(* Logix 5000 project; controller Transcat_L33ER vendor 1 type 14 code 107 rev 32.11; software revision 32.02 *)
// Upgraded CPLX to handle up to 32 EIP Nodes

TASK MainTask (continuous, watchdog 500 ms) : MainProgram

MODULES
   Local : vendor 1 type 14 code 107 (Compact 0, rev 32.11)
      GF201_Bentonite_Feeder : PowerFlex 525-EENET (Ethernet 192.168.1.195, rev 5.1, Output RPI 20 ms)   // Thayer Weigh Belt Feeder
      MX101_UpperHowesVFD : PowerFlex 525-EENET (Ethernet 192.168.1.191, rev 5.1, Output RPI 20 ms)   // VFD for Upper Howes Mixer
           MX101_UpperHowesVFD:I.Faulted   // UpperHowes Drive Faulted
           MX101_UpperHowesVFD:I.DriveStatus.4   // 1 = Accelerating
           MX101_UpperHowesVFD:I.Ready   // UpperHowes Drive Ready Status
           MX101_UpperHowesVFD:I.DriveStatus.10   // 1 - parameter locked
           MX101_UpperHowesVFD:I.DriveStatus.1   // 1 = Running, 0 - Stopped
           MX101_UpperHowesVFD:I.Active   // UpperHowes Drive Active
           MX101_UpperHowesVFD:I.DriveStatus.0   // 1 = Drive is Ready
           MX101_UpperHowesVFD:I.DriveStatus.8   // 1 = At Referecne Speed
           MX101_UpperHowesVFD:I.DriveStatus.3   // 1 = Rotating Forward
           MX101_UpperHowesVFD:I.DriveStatus.5   // 1= Decelerating
           MX101_UpperHowesVFD:I.DriveStatus.6   // not used
           MX101_UpperHowesVFD:I.DriveStatus.9   // 1 - Main Freq by Active Comms
           MX101_UpperHowesVFD:I.DriveStatus.7   // 1= Faulted
           MX101_UpperHowesVFD:I.DriveStatus.2   // 1 = Forward, 0 = Reverse
           MX101_UpperHowesVFD:O.Stop   // Drive Stop
           MX101_UpperHowesVFD:O.Start   // Drive Start
           MX101_UpperHowesVFD:O.FreqCommand   // Input Hz into Source A: 0-60 Hz range
      VF101_Medium_Feeder : PowerFlex 525-EENET (Ethernet 192.168.1.196, rev 5.1, Output RPI 20 ms)   // Medium Feeder
      MX201_LowerHowesVFD : PowerFlex 525-EENET (Ethernet 192.168.1.192, rev 5.1, Output RPI 20 ms)   // VFD for Lower Howes Mixer
           MX201_LowerHowesVFD:I.Faulted   // LowerHowes Drive Faulted
           MX201_LowerHowesVFD:I.Ready   // LowerHowes Drive Ready Status
           MX201_LowerHowesVFD:I.Active   // LowerHowes Drive Active
           MX201_LowerHowesVFD:O.Stop   // Drive Stop
      VF201_Small_Feeder_2 : PowerFlex 525-EENET (Ethernet 192.168.1.197, rev 5.1, Output RPI 20 ms)   // Acrison Small Feeder 2
      SBC2000_1_Acrison : ETHERNET-MODULE (Ethernet 192.168.1.150, rev 1.1, Output RPI 250 ms)   // Acrison Drive 1 to control Small Feeder 1
           SBC2000_1_Acrison:I.Data   // Ethernet Input Array
           SBC2000_1_Acrison:I.Data[1]   // PV - Feedrate - kg/hr
           SBC2000_1_Acrison:I.Data[2]   // Totalizer 1 - kg
           SBC2000_1_Acrison:I.Data[0]   // SP-FeedRate - kg/hr
           SBC2000_1_Acrison:I.Data[4]   // Hopper Level - %
           SBC2000_1_Acrison:I.Data[3]   // OT - Motor Speed - %
           SBC2000_1_Acrison:O.Data[15]   // When Command_Bits is 1, machine is running.
      Thayer1_BS : ETHERNET-MODULE (Ethernet 192.168.1.140, rev 1.1, Output RPI 50 ms)   // Thayer 1 Weight Belt Feeder
      Thayer2_BS : ETHERNET-MODULE (Ethernet 192.168.1.160, rev 1.1, Output RPI 50 ms)   // Thayer 2 Weigh Belt Feeder
      XS26_PLC_Safety_Controller : XS26 SC26 SC10 (Ethernet 192.168.1.211, rev 2.1, StandardDataDriven RPI 100 ms)   // XS26 Safety Controller in PLC cabinet
      XS26_VFD_Cabinet_Safety_Controller : XS26 SC26 SC10 (Ethernet 192.168.1.212, rev 2.1, StandardDataDriven RPI 100 ms)   // Banner XS26 Safety Controller with 3 expansion modules in VFD cabinet
      TC_Remote_IO : 1734-AENT (Ethernet 192.168.1.190, rev 6.1, Output RPI 20 ms)
         TC_8Pt_Analog_Input : vendor 1 type 115 code 210 (PointIO 1, rev 3.1, Input RPI 80 ms)
         TC_8pt_DC_Input_Sink : 1734-IB8 (PointIO 2, rev 3.1)
         TC_8pt_Digital_Output_Sourced : 1734-OB8 (PointIO 3, rev 3.1)
         TC_4pt_Relay_Output : 1734-OW4 (PointIO 4, rev 3.1)
END_MODULES

TYPE Acrison_Feeder :   // Acrison Feeder Tags
STRUCT
   AutoMan : BOOL;   // On - Auto Control - follows AutoRun bit, Off - Manaul Control - follows Manual Run bit
   ManualRun : BOOL;   // On - Runs feeder in Manual, Off - Stops feeder in manual
   AutoRun : BOOL;   // On - Runs feeder in Auto Off - Stops feeder in Auto
   Interlock : BOOL;   // Interlock bit - if on - Feeder will not run
   Output : BOOL;   // On - Feeder runs, Off Feeder stops
   Int_Status : DINT;   // 32 Status bits from feeder
   SP_HMI : REAL;   // setpoint from HMI
   SP_READ : REAL;   // setpoint read back from controller
   Enable : BOOL;   // Enable logic to run feeder
   OT_Actual_Hz : REAL;   // The current output of the VFD in Hz
   FreqHz_Real : REAL;   // The command frequency of the drive in Hz
   CycleTime : TIMER;   // running time of current cycle
   CampTime : TIMER;   // running time of current campaign / batch
   TotalTime : TIMER;   // total time the device / motor has run since last reset
   OneShots : BOOL[32];   // 32 Booleans to hold one-shots assicated with this device
   TimeRunTarget : DINT;   // Target Amount of time in seconds to run the device
   StartDelay : TIMER;   // Delay before motor start
   StartDelayms : DINT;   // Start delay in milliseconds
   TimeRunStart : BOOL;   // Bit to start and run a timed run
END_STRUCT
END_TYPE

TYPE BronkhorstFlowMeter :   // Read and write values for Bronkhorst Flow Meters
STRUCT
   SP_R : REAL;   // Set Point - FlowRate - Read - g/min - read from Flow Meter
   PV_R : REAL;   // Process Variable - FlowRate - Read - g/min
   OT_R : REAL;   // Output - PumpSpeed - Read - %
   TempC : REAL;   // Temperaure - Read - Deg C
   Density : REAL;   // Density - Read - g/liter
   Usertag : STRING;   // User Tag in Flow Meter - String
   FBNode : INT;   // Flow Bus Node # - Integer
   Model : STRING;   // Flow Meter Model #
   Serial : STRING;   // Flow Meter Serial #
   Capacity : REAL;   // Max Flow Rate of Flow Meter
   Enable : BOOL;   // Device enable bit
   AutoMan : BOOL;   // Select Auto / Manual Mode
   AutoRun : BOOL;   // On / Off in Auto Mode
   ManualRun : BOOL;   // On / Off- in Manual Mode
   Interlock : BOOL;   // Interlock Bit
   Output : BOOL;   // Output Bit for Device
   SP_HMI : REAL;   // Setpoint from HMI
   SP_W : REAL;   // Setpoint - flowrate g/min - write to Flow Meter from PLC
   Connected : BOOL;   // Is flow meter connecte to the flow bus network
   Alarm : BOOL;   // Alarm Bit - if on flow meter in ALarm Status
   Running : BOOL;   // the flow meter is running / dosing
   AlarmReset : BOOL;   // bit to toggle to reset alarm
   AlarmID : INT;   // Integer # that describes the type of Alarm
   ReadTime : INT;   // time in milliseconds to read the flow meter data
   DevPct : REAL;   // % deviation of process variable from setpoint
   CycleTime : TIMER;   // running time of current cycle
   CampTime : TIMER;   // running time of current campaign
   TotalTime : TIMER;   // total time the device / motor has run since last reset
   OneShots : BOOL[32];   // 32 Booleans to hold one-shots assicated with this device
   TimeRunTarget : DINT;   // Target Amount of time in seconds to run the device
   StartDelay : TIMER;   // Delay before motor start
   StartDelayms : DINT;   // Start delay in milliseconds
   TimeRunStart : BOOL;   // Bit to start and run a timed run
   Totalizer : REAL;   // Total dosed by flow meter since last reset
   TotalizerReset : BOOL;   // Bit to reset the totalizer (called a counter in Bronkhorst literature)
   TotalizerEnable : BOOL;   // Bit to turn the totalizer on / off
END_STRUCT
END_TYPE

TYPE Device :   // this UDT will be the template for all equipment / devices - feeders, flow meters, others and will be set up for each device to be indexed and processed via indirect addressing
STRUCT
   SP_R : REAL;   // Set Point - FlowRate - Read - g/min - read from Flow Meter
   PV_R : REAL;   // Process Variable - FlowRate - Read - g/min
   OT_R : REAL;   // Output - PumpSpeed - Read - %
   TempC : REAL;   // Temperaure - Read - Deg C
   Density : REAL;   // Density - Read - g/liter
   Usertag : STRING;   // User Tag in Flow Meter - String
   FBNode : INT;   // Flow Bus Node # - Integer
   Model : STRING;   // Flow Meter Model #
   Serial : STRING;   // Flow Meter Serial #
   Capacity : REAL;   // Max Flow Rate of Flow Meter
   Enable : BOOL;   // Device enable bit
   AutoMan : BOOL;   // Select Auto / Manual Mode
   AutoRun : BOOL;   // On / Off in Auto Mode
   ManualRun : BOOL;   // On / Off- in Manual Mode
   Interlock : BOOL;   // Interlock Bit
   Output : BOOL;   // Output Bit for Device
   SP_HMI : REAL;   // Setpoint from HMI
   SP_W : REAL;   // Setpoint - flowrate g/min - write to Flow Meter from PLC
   Connected : BOOL;   // Is flow meter connecte to the flow bus network
   Alarm : BOOL;   // Alarm Bit - if on flow meter in ALarm Status
   Running : BOOL;   // the flow meter is running / dosing
   AlarmReset : BOOL;   // bit to toggle to reset alarm
   AlarmID : INT;   // Integer # that describes the type of Alarm
   ReadTime : INT;   // time in milliseconds to read the flow meter data
   DevPct : REAL;   // % deviation of process variable from setpoint
   CycleTime : TIMER;   // running time of current cycle
   CampTime : TIMER;   // running time of current campaign
   TotalTime : TIMER;   // total time the device / motor has run since last reset
   OneShots : BOOL[32];   // 32 Booleans to hold one-shots assicated with this device
   TimedRunTarget : DINT;   // Target Amount of time in seconds to run the device
   StartDelay : TIMER;   // Delay before motor start
   StartDelayms : DINT;   // Start delay in milliseconds
   TimeRunEnable : BOOL;   // Bit to enable / activate a timed (campaign timed) run
   Totalizer : REAL;   // Total dosed by flow meter since last reset
   TotalizerReset : BOOL;   // Bit to reset the totalizer (called a counter in Bronkhorst literature)
   TotalizerEnable : BOOL;   // Bit to turn the totalizer on / off
   TimedRunTargetms : DINT;   // Timed run target convered to ms for use in timers
   OutPutTest : BOOL;   // A bit to simulate output that does NOT control anything
   StartDelay_ST_Timer : FBD_TIMER;   // Start delay timer to use in stuctured text
   PermissivesAuto : BOOL;   // Bit to allow device to start in AUTO as long as all permissive conditions met
   PermissivesMan : BOOL;   // Bit to allow device to start in Manual as long as all permissive conditions met
   Error : REAL;   // % Error from SP (Positive Value = running above SP and vice versa)
   ErrorTimer : TIMER;   // Amont of consecutive seconds the Error is permitterd to be out of range (+/- x%) before triggering interlock
   ErrorLimit : REAL;   // + / - % error range the system can operate in
END_STRUCT
END_TYPE

TYPE Howes_Mixer :   // Howes Mixer Tags
STRUCT
   AutoMan : BOOL;   // On - Auto Control - follows AutoRun bit, Off - Manaul Control - follows Manual Run bit
   ManualRun : BOOL;   // On - Runs feeder in Manual, Off - Stops feeder in manual
   AutoRun : BOOL;   // On - Runs feeder in Auto Off - Stops feeder in Auto
   Interlock : BOOL;   // Interlock bit - if on - Feeder will not run
   Output : BOOL;   // On - Feeder runs, Off Feeder stops
   Int_Status : DINT;   // 32 Status bits from feeder
   SP_HMI : REAL;   // setpoint from HMI
   SP_READ : REAL;   // setpoint read back from controller
   Enable : BOOL;   // Enable logic to run mixer
   FreqHz_Real : REAL;   // Frequency in Hz expressed as real #
   OT_Actual_Hz : REAL;   // The current output of the drive in Hz
   CycleTime : TIMER;   // currnet cycle run time
   CampTime : TIMER;   // current campaign run time
   TotalTime : TIMER;   // total run time since last reset
   OneShots : BOOL[32];   // 32 Booleans to hold one shots associated with this device
   TimeRunTarget : DINT;   // Target Amount of time in seconds to run the device
   TimeRunStart : BOOL;   // Bit to start and run a timed run
   StartDelay : TIMER;   // Delay before motor starts
   StartDelayms : DINT;   // Delay before motor starts in milliseconds
   RPM : REAL;   // RPM from speed sensor
END_STRUCT
END_TYPE

TYPE Thayer_WB_Feeder :   // Thayer WB Feeder Tags
STRUCT
   AutoMan : BOOL;   // On - Auto Control - follows AutoRun bit, Off - Manaul Control - follows Manual Run bit
   ManualRun : BOOL;   // On - Runs feeder in Manual, Off - Stops feeder in manual
   AutoRun : BOOL;   // On - Runs feeder in Auto Off - Stops feeder in Auto
   Interlock : BOOL;   // Interlock bit - if on - Feeder will not run
   Output : BOOL;   // On - Feeder runs, Off Feeder stops
   Int_Status : DINT;   // 32 Status bits from feeder
   SP_HMI : REAL;   // setpoint from HMI
   SP_READ : REAL;   // setpoint read back from controller
   Enable : BOOL;   // Enable logic to run feeder
   CycleTime : TIMER;   // current cycle run time
   CampTime : TIMER;   // current campaing run time
   TotalTime : TIMER;   // total run time since last reset
   OneShots : BOOL[32];   // 32 Booleans to hold one-shots assicated with this device
   TimeRunTarget : DINT;   // Target Amount of time in seconds to run the device - from recipe
   StartDelay : TIMER;   // Delay before starting motor / equipment
   StartDelayms : DINT;   // Start delay in milliseconds
   TimeRunStart : BOOL;   // Bit to start and run a timed run
END_STRUCT
END_TYPE

VAR_GLOBAL   (* controller tags *)
   AcrisonFeedRateSetPoint : MESSAGE;   // Message Command to Write to Feed Rate Set Point in Acrison from GF103.SP_HMI in kg/hr
        MessageParameters(ServiceCode := 16#0010, LocalElement := GF301.SP_HMI, ...)
   AllDevice1stScanDone : BOOL := 1;   // When this bit is set - all devices have been scanned once and bits reset
   AllDeviceEnable : BOOL := 1;   // A bit to enable or disable the running of all devices
   AllReset : BOOL;   // Bit to reset Auto/Man, AutoRun, RecipeRun, TimedRunEnable to 0 from PLC
   alwaysOFF : BOOL;
   AlwaysOFF2 : BOOL;
   AlwaysOn : BOOL;
   AnyAutoRun : BOOL;   // Bit that in on if ANY device is placed into Auto run (to signal pre-start beed)
   AnyAutoRunFlag : BOOL;   // A flag that indicates if any device is in Auto Run (used with pre-start beep logic)
   AnyManRunFlag : BOOL;   // A flag that indicates if any device is in Manual Run (used with pre-start beep logic)
   AnyManualRun : BOOL;   // Bit that in on if ANY device is placed into manual run (to signal pre-start beed)
   AnyRun : BOOL := 1;   // Bit that is true if any Maunal Run or Auto Run bit is set
   AnyRunFlag : BOOL;   // A Flag to know if any device in already running in Auto or Manual
   BeaconBeepAlarm : BOOL;   // Beep Alarm
   BeaconBlueLight : ALIAS FOR TC_Remote_IO:3:O.3;   // Blue Beacon Light
   BeaconGreenLight : ALIAS FOR TC_Remote_IO:3:O.2;   // Green Beacon Light
   BeaconRedLight : ALIAS FOR TC_Remote_IO:3:O.0;   // Red Beacon Light
   BeaconYellowLight : ALIAS FOR TC_Remote_IO:3:O.1;   // Yellow Beacon Light
   Beep : BOOL;   // Bit to Activte Beacon Alarm
   BeepNew : ALIAS FOR TC_Remote_IO:3:O.4;
   Device : Device[20] := ([0].SP_HMI := 10.6, [0].CycleTime.PRE := 288000000, [0].CycleTime.ACC := 731171, [0].CampTime.PRE := 288000000, [0].CampTime.ACC := 20003, [0].TotalTime.PRE := 288000000, [0].TotalTime.ACC := 11616964, [0].OneShots[4] := 1, [0].TimedRunTarget := 20, [0].StartDelay.PRE := 2000, [0].StartDelayms := 2, [0].TimedRunTargetms := 20000, [0].StartDelay_ST_Timer.TimerEnable := 1, [0].StartDelay_ST_Timer.PRE := 10000, [0].ErrorTimer.PRE := 10000, [1].SP_HMI := 10.6, [1].CycleTime.PRE := 288000000, [1].CycleTime.ACC := 730212, [1].CampTime.PRE := 288000000, [1].CampTime.ACC := 20004, [1].TotalTime.PRE := 288000000, [1].TotalTime.ACC := 7079420, [1].OneShots[4] := 1, [1].TimedRunTarget := 20, [1].StartDelay.PRE := 2000, [1].StartDelayms := 2, [1].TimedRunTargetms := 20000, [1].ErrorTimer.PRE := 60000, [2].CycleTime.PRE := 288000000, [2].CycleTime.ACC := 173670, [2].CampTime.PRE := 288000000, [2].CampTime.ACC := 5003, [2].TotalTime.PRE := 288000000, [2].TotalTime.ACC := 2719384, [2].OneShots[4] := 1, [2].TimedRunTarget := 5, [2].StartDelay.PRE := 2000, [2].StartDelayms := 2, [2].TimedRunTargetms := 5000, [2].PermissivesAuto := 1, [2].PermissivesMan := 1, [3].CycleTime.PRE := 288000000, [3].CycleTime.ACC := 2659, [3].CampTime.PRE := 288000000, [3].TotalTime.PRE := 288000000, [3].TotalTime.ACC := 109408498, [3].OneShots[4] := 1, [3].TimedRunTarget := 10, [3].StartDelay.PRE := 2000, [3].StartDelayms := 2, [3].TimedRunTargetms := 10000, [3].PermissivesAuto := 1, [3].PermissivesMan := 1, [4].CycleTime.PRE := 288000000, [4].CycleTime.ACC := 79705, [4].CampTime.PRE := 288000000, [4].TotalTime.PRE := 288000000, [4].TotalTime.ACC := 440481, [4].OneShots[4] := 1, [4].StartDelay.PRE := 2000,
        [4].StartDelayms := 2, [4].PermissivesAuto := 1, [4].PermissivesMan := 1, [5].CycleTime.PRE := 288000000, [5].CycleTime.ACC := 174455, [5].CampTime.PRE := 288000000, [5].CampTime.ACC := 39951, [5].TotalTime.PRE := 288000000, [5].TotalTime.ACC := 3397807, [5].OneShots[4] := 1, [5].TimedRunTarget := 120, [5].StartDelay.PRE := 2000, [5].StartDelayms := 2, [5].TimedRunTargetms := 120000, [5].PermissivesAuto := 1, [5].PermissivesMan := 1, [6].CycleTime.PRE := 288000000, [6].CycleTime.ACC := 485, [6].CampTime.PRE := 288000000, [6].CampTime.ACC := 39952, [6].TotalTime.PRE := 288000000, [6].TotalTime.ACC := 3344121, [6].OneShots[4] := 1, [6].TimedRunTarget := 120, [6].StartDelay.PRE := 2000, [6].StartDelayms := 2, [6].TimedRunTargetms := 120000, [6].PermissivesAuto := 1, [6].PermissivesMan := 1, [7].SP_HMI := 150.0, [7].CycleTime.PRE := 288000000, [7].CycleTime.ACC := 39946, [7].CampTime.PRE := 288000000, [7].CampTime.ACC := 39951, [7].TotalTime.PRE := 288000000, [7].TotalTime.ACC := 8389325, [7].OneShots[4] := 1, [7].TimedRunTarget := 120, [7].StartDelay.PRE := 5000, [7].StartDelayms := 5, [7].TimedRunTargetms := 120000, [8].CycleTime.PRE := 288000000, [8].CycleTime.ACC := 39947, [8].CampTime.PRE := 288000000, [8].CampTime.ACC := 39952, [8].TotalTime.PRE := 288000000, [8].TotalTime.ACC := 7574006, [8].OneShots[4] := 1, [8].TimedRunTarget := 120, [8].StartDelay.PRE := 5000, [8].StartDelayms := 5, [8].TimedRunTargetms := 120000, [9].CycleTime.PRE := 288000000, [9].CycleTime.ACC := 39946, [9].CampTime.PRE := 288000000, [9].CampTime.ACC := 39951, [9].TotalTime.PRE := 288000000, [9].TotalTime.ACC := 6215395, [9].OneShots[4] := 1, [9].TimedRunTarget := 120,
        [9].StartDelay.PRE := 5000, [9].StartDelayms := 5, [9].TimedRunTargetms := 120000, [10].CycleTime.PRE := 288000000, [10].CampTime.PRE := 288000000, [10].TotalTime.PRE := 288000000, [10].OneShots[2] := 1, [10].OneShots[4] := 1, [11].CycleTime.ACC := 6, [11].CycleTime.DN := 1, [11].TotalTime.ACC := 7, [11].TotalTime.DN := 1, [11].OneShots[4] := 1, [11].PermissivesAuto := 1, [11].PermissivesMan := 1);
        [8]   // FT104 - Bronkhorst Water Dosing System
        [9]   // FT105 Bronkhorst Fragrance Dosing System
        [4]   // GF301 Small Feeder - Acrison LIW
        [0]   // MX101 - Upper Howes Mixer
        [1]   // MX201 - Lower Howes Mixer
        [2]   // GF101 - Thayer1 WB Feeder
        [3]   // GF201 - Thayer2 WB Feeder
        [5]   // VF101 Medium Feeder - Acurate
        [7]   // FT103 - Bronkhorst Oil Dosing System
        [6]   // VF201 Small Feeder 2 - Acrison
   DINT_Temp : DINT;   // Place to hold Dint's durng transition to new PLC
   DiscreteTemp : BOOL;   // A temporay boolean to hold positions during PLC transer
   dNum : INT := 1;   // The index of the current device being processed
   DoseCounter : COUNTER := (ACC := 522, CU := 1, DN := 1);   // Counts the # of doses since last reset
   DoseCounterReset_HMI : BOOL;   // HMI bit to reset the dose counter
   DoseStart : BOOL;   // Bit to start dosing sequence
   DoseStartOneShot : BOOL := 1;   // One shot to start dosing
   DoseStop : BOOL;   // Bit to stop dosing
   DoseStopOneShot : BOOL := 1;   // one shot to stop dosing
   DoseTarget : REAL := 27.9;   // Target dose amount
   FT103 : BronkhorstFlowMeter := (Usertag := 'FT-103', Model := 'M55-RGD-25-0-S', Serial := 'M22213015A', Capacity := 1000.00006, Enable := 1, SP_HMI := 50.0, ReadTime := 500, CycleTime.PRE := 288000000, CycleTime.ACC := 19487, CampTime.PRE := 28800000, CampTime.ACC := 10001, TotalTime.PRE := 999999999, TotalTime.ACC := 114629);
   FT104 : BronkhorstFlowMeter := (PV_R := -97.77293, TempC := 21.284956, Density := 9999.0, Usertag := 'FT-104          ', Model := 'M55-RGD-25-0-S', Serial := 'M22213015C', Capacity := 10000.0, Enable := 1, SP_HMI := 100.0, Connected := 1, ReadTime := 70, CycleTime.PRE := 288000000, CycleTime.ACC := 3248, CampTime.PRE := 28800000, CampTime.ACC := 10001, TotalTime.PRE := 999999999, TotalTime.ACC := 84417, StartDelay.PRE := 2000, StartDelayms := 2);
   FT105 : BronkhorstFlowMeter := (PV_R := 0.458107, TempC := 28.406788, Density := 4.5310874, Usertag := 'FT-105          ', Model := 'M14-RGD-22-0-S', Serial := 'M20210127A', Capacity := 202.79999, Enable := 1, SP_HMI := 75.0, Connected := 1, ReadTime := 64, CycleTime.PRE := 288000000, CycleTime.ACC := 11357, CampTime.PRE := 28800000, CampTime.ACC := 10001, TotalTime.PRE := 999999999, TotalTime.ACC := 55929, StartDelay.PRE := 4000, StartDelayms := 4);
   GF101 : Thayer_WB_Feeder := (SP_HMI := 21.4, SP_READ := 21.375, Enable := 1, CycleTime.PRE := 288000000, CycleTime.ACC := 9195, CampTime.PRE := 28800000, CampTime.ACC := 10001, TotalTime.PRE := 999999999, TotalTime.ACC := 1761327, StartDelay.PRE := 2000, StartDelayms := 2);   // Thayer 1 Tags
   GF101_Alarm_ExcessDevSP : ALIAS FOR Thayer1_BS:I.Data[8].7;   // Thayer 1 (GF101) - Alarm - excessive deviation from SP
   GF101_LoadCell : ALIAS FOR Thayer1Data[15];   // Thayer 1 (GF101) load cell in lbs
   GF101_LoadCellTempF : ALIAS FOR Thayer1Data[16];   // Thayer 1 (GF101) load cell temperature in Deg F
   GF101_OutputPct : ALIAS FOR Thayer1Data[5];   // Thayer 1 (GF101) Output to motor in pct - raw
   GF101_RunningLoad : ALIAS FOR Thayer1Data[0];   // Thayer 1 (GF101) Running Load - current load on belt in lbs
   GF101_RunningRate : ALIAS FOR Thayer1Data[1];   // Thayer 1 (GF101) Running Rate - current PV displayed on the operator screen
   GF101_RunningSpeed : ALIAS FOR Thayer1Data[2];   // Thayer 1 (GF101) Running Soeed - current speed of the belt in ft/min?
   GF101_SetPoint : ALIAS FOR Thayer1Data[3];   // Thayer 1 (GF101) SetPoint - in lb/min
   GF101_Shutdown_ExcessDevSp : ALIAS FOR Thayer1_BS:I.Data[10].7;   // Thayer 1 (GF101) - Shutdown - excessive deviation from SP
   GF101_Status_AutoMan : ALIAS FOR Thayer1_BS:I.Data[0].1;   // Thayer 1 (GF101) - Auto / Manual Status - 1 = Auto 0 = Manual
   GF101_Status_Coasting : ALIAS FOR Thayer1_BS:I.Data[0].2;   // Thayer 1 (GF101) - Coasting to stop of shutdown - 1 = Coasting, 0 = Not coasting
   GF101_Status_EchoBack : ALIAS FOR Thayer1_BS:I.Data[0].13;   // Thayer 1 (GF101) - Echo back bit
   GF101_Status_HeartBeat : ALIAS FOR Thayer1_BS:I.Data[0].14;   // Thayer 1 (GF101) - HeartBeat - every 5 seconds
   GF101_Status_Interlocked : ALIAS FOR Thayer1_BS:I.Data[0].8;   // Thayer 1 (GF101) - Interlocked Bit - 1 = Interlocked 0 = Not Interlocked
   GF101_Status_RunStop : ALIAS FOR Thayer1_BS:I.Data[0].0;   // Thayer 1 (GF101) - Operating Status - 1 = Running 0 = Stopped
   GF101_Status_TachGT0 : ALIAS FOR Thayer1_BS:I.Data[0].9;   // Thayer 1 (GF101) - 1 = Tachometer > 0 0 = Tachometer = 0
   GF101_TachHz : ALIAS FOR Thayer1Data[14];   // Thayer 1 (GF101) Tachometer in Hz
   GF101_Totalizer1 : ALIAS FOR Thayer1Data[9];   // Thayer 1 (GF101) Totalizer 1 in lbs
   GF101_Totalizer2 : ALIAS FOR Thayer1Data[10];   // Thayer 1 (GF101) Totalizer 2 in lbs
   GF101_Write_Acknowledge : ALIAS FOR Thayer1_BS:O.Data[2].5;   // Thayer 1 (GF101) Acknowledge
   GF101_Write_AutoMan : ALIAS FOR Thayer1_BS:O.Data[0].1;   // Thayer 1 (GF101) Auto / Manual 1 = Auto 2 = Manual
   GF101_Write_RunStop : ALIAS FOR Thayer1_BS:O.Data[0].0;   // Thayer 1 (GF101) 1 = Run / 0 = off/stop
   GF101_Write_Total1Reset : ALIAS FOR Thayer1_BS:O.Data[2].1;   // Thayer 1 (GF101) Totalizer 1 reset
   GF101_Write_Total2Reset : ALIAS FOR Thayer1_BS:O.Data[2].2;   // Thayer 1 (GF101) Totalizer 2 reset
   GF101OutpuyPct1sec : ALIAS FOR Thayer1Data[6];   // Thayer 1 (GF101) Output to motor in pct - averaged over 1 sec
   GF201 : Thayer_WB_Feeder := (SP_HMI := 20.0, SP_READ := 20.0, Enable := 1, CycleTime.PRE := 288000000, CycleTime.ACC := 17126, CampTime.PRE := 28800000, CampTime.ACC := 10001, TotalTime.PRE := 999999999, TotalTime.ACC := 1645614, StartDelay.PRE := 2000, StartDelayms := 2);   // Thayer 2 Tags
   GF201_Alarm_ExcessiDevSP : ALIAS FOR Thayer2_BS:I.Data[8].7;   // Thayer 2 (GF201) - Alarm - excessive deviation from SP
   GF201_LoadCell : ALIAS FOR Thayer2Data[15];   // Thayer 2 (GF201) load cell in lbs
   GF201_LoadCellTempF : ALIAS FOR Thayer2Data[16];   // Thayer 2 (GF201) load cell temperature in Deg F
   GF201_OutputPct : ALIAS FOR Thayer2Data[5];   // Thayer 2 (GF201) Output to motor in pct - raw
   GF201_RunningLoad : ALIAS FOR Thayer2Data[0];   // Thayer 2 (GF201) Running Load - current load on belt in lbs
   GF201_RunningRate : ALIAS FOR Thayer2Data[1];   // Thayer 2 (GF201) Running Rate - current PV displayed on the operator screen
   GF201_RunningSpeed : ALIAS FOR Thayer2Data[2];   // Thayer 2 (GF201) Running Soeed - current speed of the belt in ft/min?
   GF201_SetPoint : ALIAS FOR Thayer2Data[3];   // Thayer 2 (GF201) SetPoint - in lb/min
   GF201_Shutdown_ExcessDevSP : ALIAS FOR Thayer2_BS:I.Data[10].7;   // Thayer 2 (GF201) - Shutdown - excessive deviation from SP
   GF201_Status_AutoMan : ALIAS FOR Thayer2_BS:I.Data[0].1;   // Thayer 2 (GF201) - Auto / Manual Status - 1 = Auto 0 = Manual
   GF201_Status_Coasting : ALIAS FOR Thayer2_BS:I.Data[0].2;   // Thayer 2 (GF201) - Coasting to stop of shutdown - 1 = Coasting, 0 = Not coasting
   GF201_Status_EchoBack : ALIAS FOR Thayer2_BS:I.Data[0].13;   // Thayer 2 (GF201) - Echo back bit
   GF201_Status_HeartBeat1 : ALIAS FOR Thayer2_BS:I.Data[0].14;   // Thayer 2 (GF201) - HeartBeat - every 5 seconds
   GF201_Status_Interlocked : ALIAS FOR Thayer2_BS:I.Data[0].8;   // Thayer 2 (GF201) - Interlocked Bit - 1 = Interlocked 0 = Not Interlocked
   GF201_Status_RunStop : ALIAS FOR Thayer2_BS:I.Data[0].0;   // Thayer 2 (GF201) - Operating Status - 1 = Running 0 = Stopped
   GF201_Status_TachGT0 : ALIAS FOR Thayer2_BS:I.Data[0].9;   // Thayer 2 (GF201) - 1 = Tachometer > 0 0 = Tachometer = 0
   GF201_TachHz : ALIAS FOR Thayer2Data[14];   // Thayer 2 (GF201) Tachometer in Hz
   GF201_Totalizer1 : ALIAS FOR Thayer2Data[9];   // Thayer 2 (GF201) Totalizer 1 in lbs
   GF201_Totalizer2 : ALIAS FOR Thayer2Data[10];   // Thayer 2 (GF201) Totalizer 2 in lbs
   GF201_Write_Acknowledge : ALIAS FOR Thayer2_BS:O.Data[2].5;   // Thayer 2 (GF201) Acknowledge
   GF201_Write_AutoMan : ALIAS FOR Thayer2_BS:O.Data[0].1;   // Thayer 2 (GF201) Auto / Manual 1 = Auto 2 = Manual
   GF201_Write_RunStop : ALIAS FOR Thayer2_BS:O.Data[0].0;   // Thayer 2 (GF201) 1 = Run / 0 = off/stop
   GF201_Write_Total1Reset : ALIAS FOR Thayer2_BS:O.Data[2].1;   // Thayer 2 (GF1201) Totalizer 1 reset
   GF201_Write_Total2Reset : ALIAS FOR Thayer2_BS:O.Data[2].2;   // Thayer 2 (GF201) Totalizer 2 reset
   GF201OutpuyPct1sec : ALIAS FOR Thayer2Data[6];   // Thayer 2 (GF201) Output to motor in pct - averaged over 1 sec
   GF301 : Acrison_Feeder := (Int_Status := 596060, SP_HMI := 8.0, Enable := 1, CycleTime.PRE := 288000000, CycleTime.ACC := 223848, CampTime.PRE := 28800000, CampTime.ACC := 10001, TotalTime.PRE := 999999999, TotalTime.ACC := 2086091, StartDelay.PRE := 2000, StartDelayms := 2);   // GF103 - Small Feeder 1
        .Int_Status.3   // SP Int-1 / Ext-0
        .Int_Status.5   // Batch-1 / Cont-0
        .Int_Status.11   // Alarm
        .Output   // GF103 - Acrison Small Feeder Run Bit
        .Int_Status.13   // Empty
        .Int_Status.4   // Mode - Grav-1 / Vol-0
        .Int_Status.17   // Deviation
        .Int_Status.12   // Message
        .Int_Status.14   // Overfill
        .Int_Status.15   // Acrilock
        .Int_Status.16   // No Scale
        .Int_Status.10   // Overfill / Empty
        .Int_Status.1   // Refil
        .Int_Status.2   // AutoRefill
        .Int_Status.7   // Bribble
        .Int_Status.0   // Run-1 / Stop-0
        .Int_Status.9   // Low Level
        .Int_Status.6   // Batch Complete
        .Int_Status   // 32 Bit Status Int
        .Int_Status.8   // High Level
   GF301_AlarmAck : BOOL;   // GF301 Alarm Ack Bit
   GF301_ClearCommands : BOOL;   // Bit to send clear command to GF301 command integer
   GF301_Command_Bits : INT;   // Command Word - Holds a value that gets written to Acrison SCB2000:I.Data[15] see Acrison Manual for which bits do what
        .1   // Refill Mode Man - 1 / Auto - 0
        .0   // Run-1 / Stop-0
        .8   // Setpoint - Ext -1 / Int - 0
        .2   // Batch-1 / Cont-0
        .4   // Refill ON
        .6   // Alarm Ack
        .5   // Refill OFF
        .3   // Batch Abort
        .7   // Mode Vol - 1/ Grav - 0
   GF301_IntStatus : DINT := 596060;   // 32 Bit Status INT for GF301
        .14   // Overfill
        .12   // Message
        .10   // Overfill / Empty
        .0   // Run- 1/ Stop - 0
        .15   // Acrilok
        .6   // Batch Complete
        .9   // Low Level
        .16   // No Scale
        .3   // Setpoint Int - 1 / Ext - 0
        .17   // Deviation
        .1   // Refil
        .2   // Auto Refill
        .4   // Mode Grav - 1 / Vol - 0
        .11   // Alarm
        .8   // High Level
        .13   // Empty
        .7   // Dribble
        .5   // Batch - 1 / Cont - 0
   GF301_OT : ALIAS FOR SBC2000_1_Acrison:I.Data[3];   // GF301 Ouput ot motor in %
   GF301_PV : ALIAS FOR SBC2000_1_Acrison:I.Data[1];   // GF301 PV - Process Variable
   GF301_SP_READ : ALIAS FOR SBC2000_1_Acrison:I.Data[0];   // GF301 Set point read back from Acrison - kg/min
   GF301_TOTAL : ALIAS FOR SBC2000_1_Acrison:I.Data[2];   // GF301 Totalizer in KG
   GreenFlashingOff : TIMER := (PRE := 500);
   GreenFlashingOn : TIMER := (PRE := 500);
   HertzSetting : ALIAS FOR MX101_UpperHowesVFD:O.FreqCommand.0;   // UserHzSetting
   HMI_AllReset : BOOL;   // Bit to reset Auto/Man, AutoRun, RecipeRun, TimedRunEnable to 0 from HMI
   HMI_RecipeStart : BOOL;   // Bit to start and stop recipe from HMI
   InitCount : INT := 10;   // Counter to cycle through each device on start-up and reset AutoMan, AutoRun, ManualRun bits
   MSG_FROM_SLC500 : INT[10] := ([1] := 2500, [2] := 200, [3] := 300, [4] := 400, [5] := 500, [6] := 16, [7] := 17, [8] := 18, [9] := 19); {produced}
   MX101 : Howes_Mixer := (AutoMan := 1, SP_HMI := 120.0, Enable := 1, FreqHz_Real := 40.0, CycleTime.PRE := 288000000, CycleTime.ACC := 4243, CampTime.PRE := 28800000, CampTime.ACC := 10001, TotalTime.PRE := 999999999, TotalTime.ACC := 1803981, TimeRunTarget := 10000, StartDelay.PRE := 2000, StartDelayms := 2, RPM := -0.09);
   MX101_RPM_RAW : ALIAS FOR Test_Hold;   // Raw (unscaled) RMS reading from MX101 speed sensor - RPM * 100 (range 0 - 200 RPM)
   MX101_Speed_Hold : DINT := 100;   // Constant Value for MX101 RPM meter - till Actual signal comes back from 4-20mA from sensor
   MX201 : Howes_Mixer := (AutoMan := 1, SP_HMI := 120.0, Enable := 1, FreqHz_Real := 40.0, CycleTime.PRE := 28800000, CycleTime.ACC := 117513, CampTime.PRE := 28800000, CampTime.ACC := 10001, TotalTime.PRE := 999999999, TotalTime.ACC := 1030054, TimeRunTarget := 10000, StartDelay.PRE := 2000, StartDelayms := 2, RPM := -0.06);
   MX201_RPM_RAW : ALIAS FOR Test_Hold;   // Raw (unscaled) RMS reading from MX201 speed sensor - RPM * 100 (range 0 - 200 RPM)
   MX201_Speed_Hold : DINT := 100;   // Constant Value for MX201 RPM meter - till Actual signal comes back from 4-20mA from sensor
   PowerOffThayer1 : BOOL;
   PowerOnThayer1 : BOOL;
   PT103_HP_Interlock : BOOL;
   PT103_PV_RAW : ALIAS FOR TC_Remote_IO:1:I.Ch0Data;   // Raw (unscaled) pressure reading from PT103 - PSI * 100 (range 0 - 108 PSI)
   PT104_PV_RAW : ALIAS FOR TC_Remote_IO:1:I.Ch1Data;   // Raw (unscaled) pressure reading from PT104 - PSI * 100 (range 0 - 108 PSI)
   PT105_PV_RAW : ALIAS FOR TC_Remote_IO:1:I.Ch2Data;   // Raw (unscaled) pressure reading from PT105 - PSI * 100 (range 0 - 108 PSI)
   RandomFloat : REAL[20] := ([0] := 324.0, [1] := 11268015.0, [2] := 20.713356, [3] := 16.079597, [4] := 74.3938, [5] := 86.28061, [6] := 69.73996, [7] := 47.361, [8] := 43.876316, [9] := 89.62069, [10] := 12.1234);
   RandomSeed : DINT := 258;
   RandomTimer : TIMER := (PRE := 1000, ACC := 146, EN := 1, TT := 1);
   RecipeStart : BOOL;   // Bit to start and stop a recipe execution from PLC logic
   rms : BOOL;
   StartBeepTimer : TIMER := (PRE := 2500);   // Timer to sound the beep alarm before starting a device
   TempReal1 : REAL;
   Test_Hold : DINT;   // Place for RPM and Pressure sensors to Alias for while the AI's are not available
   TestBit1 : BOOL;   // Just a test bit - does not do anything
   Thayer1_SP : REAL := 20.0;
   Thayer1Ackn_SilenceRequest : BOOL;
   Thayer1Automatic : BOOL;
   Thayer1Data : REAL[40] := ([0] := 11.25, [1] := 1.4906e-41, [3] := 21.375, [4] := 2.0, [9] := 580.0, [10] := 583.5728, [11] := 8.2028e-41, [15] := 11.25, [16] := 70.58101, [17] := 1.6071e-41, [19] := 11.25);
        [10]   // Totalizer 2
        [11]   // take a way totalizer - not used
        [2]   // Running Speed - belt speed in ft / min
        [1]   // Running Rate - Process variable in lb/min
        [7]   // not used
        [9]   // Totalizer 1
        [0]   // Running Load - load cell reading in lbs
        [15]   // Load Cell reading lbs.
        [14]   // Tachometer - Hz
        [3]   // SetPoint - in lb/min
        [8]   // not used
        [6]   // Drive Output in % (1 sec time averaged)
        [4]   // Ratio Setpoint - not used
        [5]   // Drive Output in %
        [12]   // take away belt load - not used
        [16]   // Load Cell Temperatue - Deg F
        [17]   // Auto Zero error log in %
        [13]   // Take away belt rate - not used
   Thayer1PowerOn : BOOL;
   Thayer1ResetTotalizers : BOOL;
   Thayer1SetPoint : REAL[1];
   Thayer1SpeedControl : REAL := 20.0;
   Thayer2_SP : REAL := 20.0;
   Thayer2Automatic : BOOL;
   Thayer2Data : REAL[40] := ([0] := 7.3125, [1] := 3.7907e-41, [3] := 20.0, [9] := 0.91015625, [10] := 15288.634, [11] := 7.6957e-41, [15] := 7.3125, [16] := 70.7114, [17] := 1.6071e-41, [19] := 7.3125);
   Thayer2PowerOn : BOOL;
   Thayer2ResetTotal1_HMI : BOOL;   // Bit to reset Thayer2 - totalizer 1 from HMI
   Thayer2ResetTotalizers : BOOL;
   Thayer2SpeedControl : REAL := 20.0;
   TotalRestOneShot : BOOL;   // one shot for total reset
   UHStartOneShot : BOOL;
   UHStopOneShot : BOOL;
   UpHowesHMIRun : BOOL;
   UpHowesHMIStop : BOOL;
   UpHowesSpeedHMI : INT;
   UpperHowesSpeed : INT := 2500;
   UpperHowesStart : BOOL;
   UpperHowesStop : BOOL;
   UserBit1 : BOOL;   // user controlled bit for testing
   VF101 : Acrison_Feeder := (SP_HMI := 16.81, Enable := 1, FreqHz_Real := 10.09, CycleTime.PRE := 288000000, CycleTime.ACC := 7359, CampTime.PRE := 28800000, CampTime.ACC := 10001, TotalTime.PRE := 999999999, TotalTime.ACC := 1720239, StartDelay.PRE := 5000, StartDelayms := 5);   // Medium Feeder Tags
   VF201 : Acrison_Feeder := (SP_HMI := 14.7, Enable := 1, FreqHz_Real := 8.82, CycleTime.PRE := 288000000, CycleTime.ACC := 13534, CampTime.PRE := 28800000, CampTime.ACC := 10001, TotalTime.PRE := 999999999, TotalTime.ACC := 1964985, StartDelay.PRE := 5000, StartDelayms := 5);   // Small Feeder 2 Tags
   YellowFlashOff : TIMER := (PRE := 500);
   YellowFlashOn : TIMER := (PRE := 500, ACC := 394, EN := 1, TT := 1);
   ZS101_RPM_Speed_UpperHowes : ALIAS FOR TC_Remote_IO:1:I.Ch3Data;   // Upper Howes Zero Speed Sensor RPM
   ZS102_RPM_Speed_LowerHowes : ALIAS FOR TC_Remote_IO:1:I.Ch4Data;   // Lower Howes Zero Speed Sensor RPM
END_VAR

PROGRAM MainProgram   (* main routine MainRoutine *)
VAR
   AcrisonSpeedControl : REAL := 1.0;
   AcrisonSpeedControl2 : REAL := 15.0;
   HertzInput : INT := 20;
   Int_Status : DINT := 540252;
   LowerHowesSpeedSensor : REAL := -74.971405;
   PowerOffACrison : BOOL := 1;
   PowerOnAcrison : BOOL;
   SCL_01 : SCALE := (In := -21.0, InRawMax := 16384.0, InRawMin := 3271.0, InEUMax := 300.0, Out := -75.314575, MinAlarm := 1);
   SCL_02 : SCALE := (In := -6.0, InRawMax := 16384.0, InRawMin := 3271.0, InEUMax := 300.0, Out := -74.971405, MinAlarm := 1);
   SpeedSensorUpperHowesSpeed : REAL := -75.314575;
   T1 : TIMER := (PRE := 10000);
   T2 : TIMER := (PRE := 10000, ACC := 10000, EN := 1, DN := 1);
END_VAR

ROUTINE Auxillary_Pump_AE   (* ladder *)
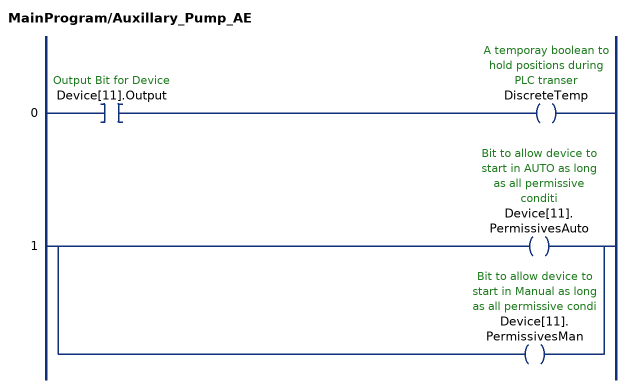
   0: XIC(Device[11].Output)OTE(DiscreteTemp);
   1: [OTE(Device[11].PermissivesAuto) ,OTE(Device[11].PermissivesMan) ];
END_ROUTINE

ROUTINE DeviceLogic   (* ladder *)
// Process the logic for each device with index and indirect addressing.
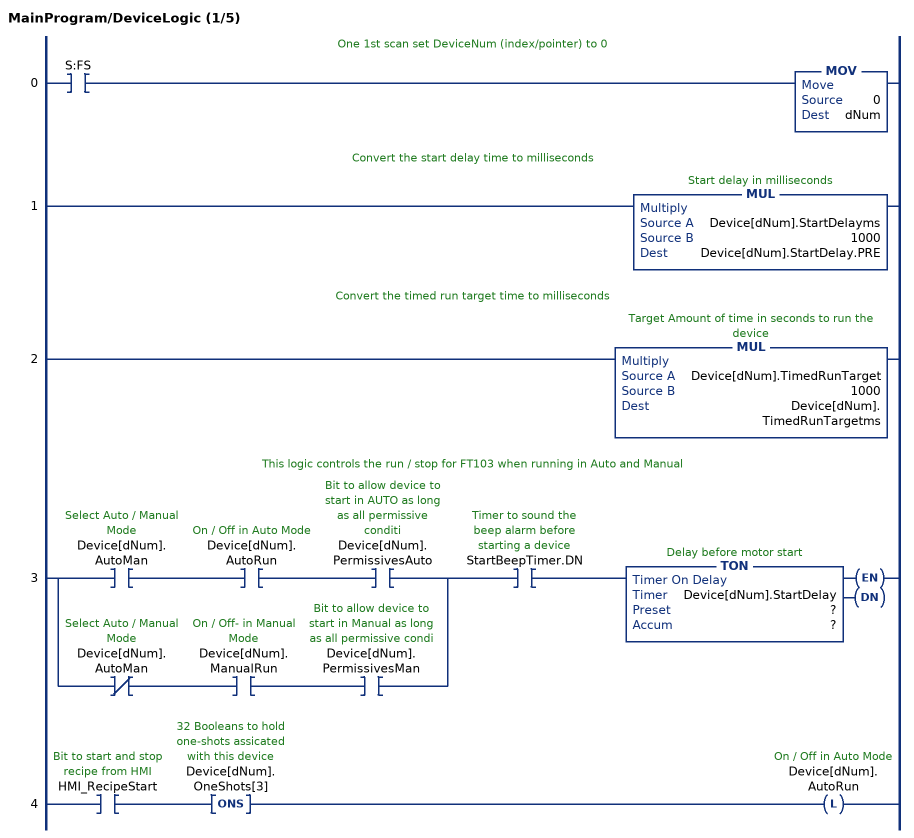
   // One 1st scan set DeviceNum (index/pointer) to 0
   0: XIC(S:FS)MOV(0,dNum);
   // Convert the start delay time to milliseconds
   1: MUL(Device[dNum].StartDelayms,1000,Device[dNum].StartDelay.PRE);
   // Convert the timed run target time to milliseconds
   2: MUL(Device[dNum].TimedRunTarget,1000,Device[dNum].TimedRunTargetms);
   // This logic controls the run / stop for FT103 when running in Auto and Manual
   3: [XIC(Device[dNum].AutoMan) XIC(Device[dNum].AutoRun) XIC(Device[dNum].PermissivesAuto) ,XIO(Device[dNum].AutoMan) XIC(Device[dNum].ManualRun) XIC(Device[dNum].PermissivesMan) ]XIC(StartBeepTimer.DN)TON(Device[dNum].StartDelay,?,?);
   4: XIC(HMI_RecipeStart)ONS(Device[dNum].OneShots[3])OTL(Device[dNum].AutoRun);
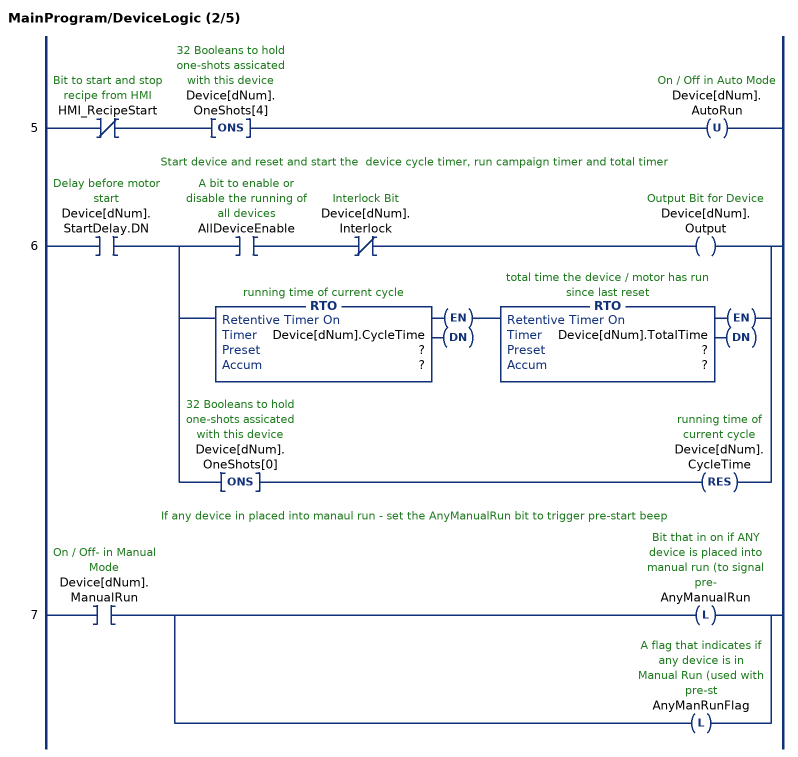
   5: XIO(HMI_RecipeStart)ONS(Device[dNum].OneShots[4])OTU(Device[dNum].AutoRun);
   // Start device and reset and start the  device cycle timer, run campaign timer and total timer
   6: XIC(Device[dNum].StartDelay.DN)[XIC(AllDeviceEnable) XIO(Device[dNum].Interlock) OTE(Device[dNum].Output) ,[RTO(Device[dNum].CycleTime,?,?) RTO(Device[dNum].TotalTime,?,?) ,ONS(Device[dNum].OneShots[0]) RES(Device[dNum].CycleTime) ] ];
   // If any device in placed into manaul run - set the AnyManualRun bit to trigger pre-start beep
   7: XIC(Device[dNum].ManualRun)[OTL(AnyManualRun) ,OTL(AnyManRunFlag) ];
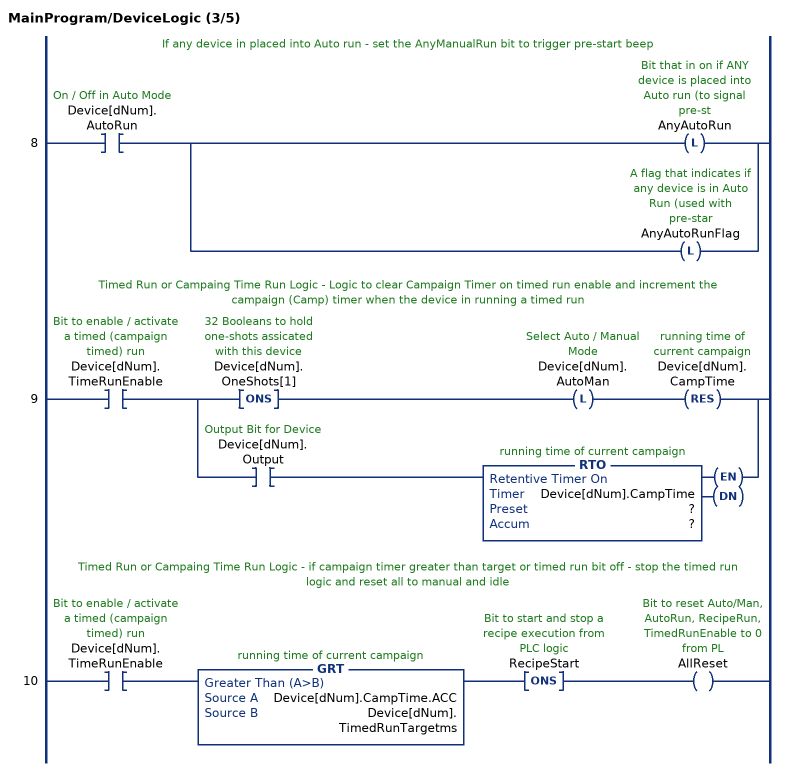
   // If any device in placed into Auto run - set the AnyManualRun bit to trigger pre-start beep
   8: XIC(Device[dNum].AutoRun)[OTL(AnyAutoRun) ,OTL(AnyAutoRunFlag) ];
   // Timed Run or Campaing Time Run Logic - Logic to clear Campaign Timer on timed run enable and increment the campaign (Camp) timer when the device in running a timed run
   9: XIC(Device[dNum].TimeRunEnable)[ONS(Device[dNum].OneShots[1]) OTL(Device[dNum].AutoMan) RES(Device[dNum].CampTime) ,XIC(Device[dNum].Output) RTO(Device[dNum].CampTime,?,?) ];
   // Timed Run or Campaing Time Run Logic - if campaign timer greater than target or timed run bit off - stop the timed run logic and reset all to manual and idle
   10: XIC(Device[dNum].TimeRunEnable)GRT(Device[dNum].CampTime.ACC,Device[dNum].TimedRunTargetms)ONS(RecipeStart)OTE(AllReset);
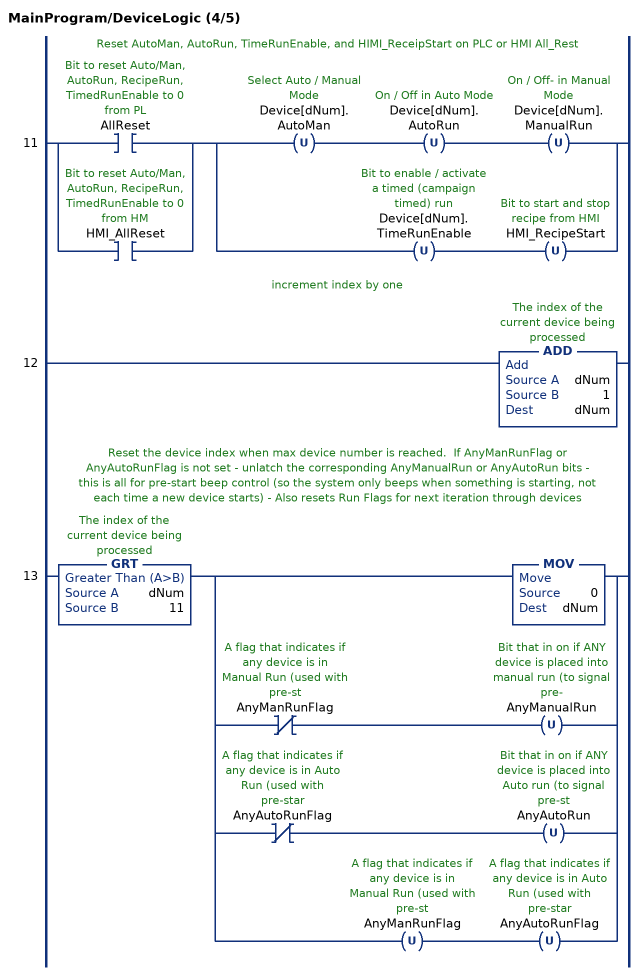
   // Reset AutoMan, AutoRun, TimeRunEnable, and HIMI_ReceipStart on PLC or HMI All_Rest
   11: [XIC(AllReset) ,XIC(HMI_AllReset) ][OTU(Device[dNum].AutoMan) OTU(Device[dNum].AutoRun) OTU(Device[dNum].ManualRun) ,OTU(Device[dNum].TimeRunEnable) OTU(HMI_RecipeStart) ];
   // increment index by one
   12: ADD(dNum,1,dNum);
   // Reset the device index when max device number is reached.  If AnyManRunFlag or AnyAutoRunFlag is not set - unlatch the corresponding AnyManualRun or AnyAutoRun bits - this is all for pre-start beep control (so the system only beeps when something is starting, not each time a new device starts) - Also resets Run Flags for next iteration through devices
   13: GRT(dNum,11)[[MOV(0,dNum) ,[XIO(AnyManRunFlag) OTU(AnyManualRun) ,XIO(AnyAutoRunFlag) OTU(AnyAutoRun) ] ] ,OTU(AnyManRunFlag) OTU(AnyAutoRunFlag) ];
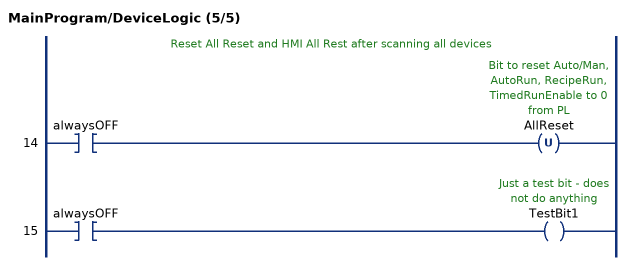
   // Reset All Reset and HMI All Rest after scanning all devices
   14: XIC(alwaysOFF)OTU(AllReset);
   15: XIC(alwaysOFF)OTE(TestBit1);
END_ROUTINE

ROUTINE FT103_Oil_Dosing   (* ladder *)
// Logic to control FT103 not associated with Device Iteration Logic
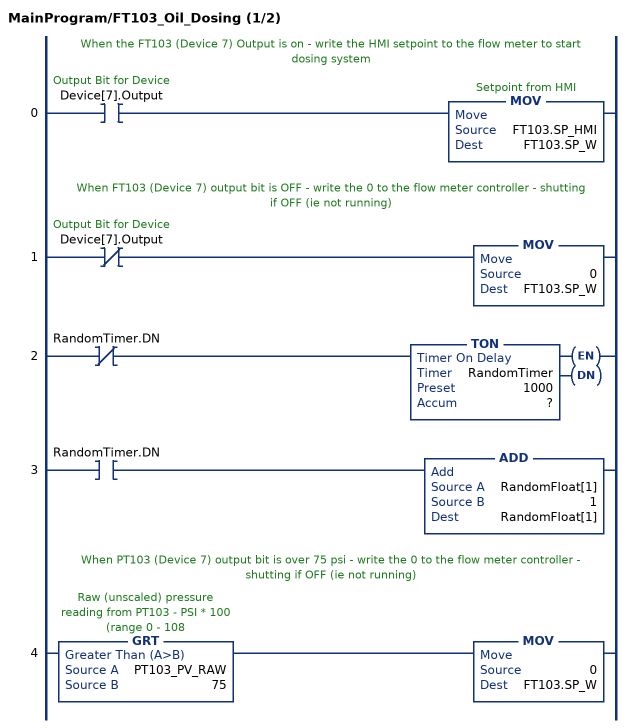
   // When the FT103 (Device 7) Output is on - write the HMI setpoint to the flow meter to start dosing system
   0: XIC(Device[7].Output)MOV(FT103.SP_HMI,FT103.SP_W);
   // When FT103 (Device 7) output bit is OFF - write the 0 to the flow meter controller - shutting if OFF (ie not running)
   1: XIO(Device[7].Output)MOV(0,FT103.SP_W);
   2: XIO(RandomTimer.DN)TON(RandomTimer,?,?);
   3: XIC(RandomTimer.DN)ADD(RandomFloat[1],1,RandomFloat[1]);
   // When PT103 (Device 7) output bit is over 75 psi - write the 0 to the flow meter controller - shutting if OFF (ie not running)
   4: GRT(PT103_PV_RAW,75)MOV(0,FT103.SP_W);
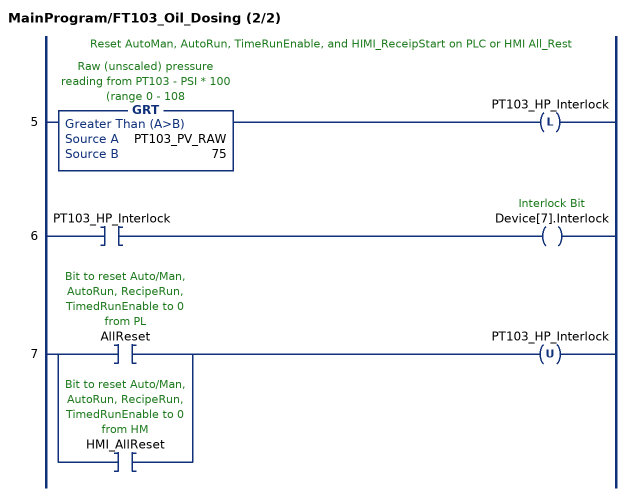
   // Reset AutoMan, AutoRun, TimeRunEnable, and HIMI_ReceipStart on PLC or HMI All_Rest
   5: GRT(PT103_PV_RAW,75)OTL(PT103_HP_Interlock);
   6: XIC(PT103_HP_Interlock)OTE(Device[7].Interlock);
   7: [XIC(AllReset) ,XIC(HMI_AllReset) ]OTU(PT103_HP_Interlock);
END_ROUTINE

ROUTINE FT104_Water_Dosing   (* ladder *)
// FT104 Control Logic not associated with Device Iteration Logic
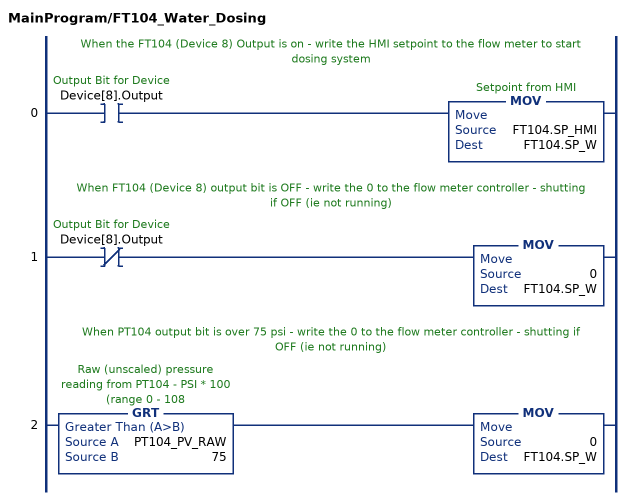
   // When the FT104 (Device 8) Output is on - write the HMI setpoint to the flow meter to start dosing system
   0: XIC(Device[8].Output)MOV(FT104.SP_HMI,FT104.SP_W);
   // When FT104 (Device 8) output bit is OFF - write the 0 to the flow meter controller - shutting if OFF (ie not running)
   1: XIO(Device[8].Output)MOV(0,FT104.SP_W);
   // When PT104 output bit is over 75 psi - write the 0 to the flow meter controller - shutting if OFF (ie not running)
   2: GRT(PT104_PV_RAW,75)MOV(0,FT104.SP_W);
END_ROUTINE

ROUTINE FT105_Fragrance_Dosing   (* ladder *)
// FT105 Control Logic not associated with Device Iteration Logic
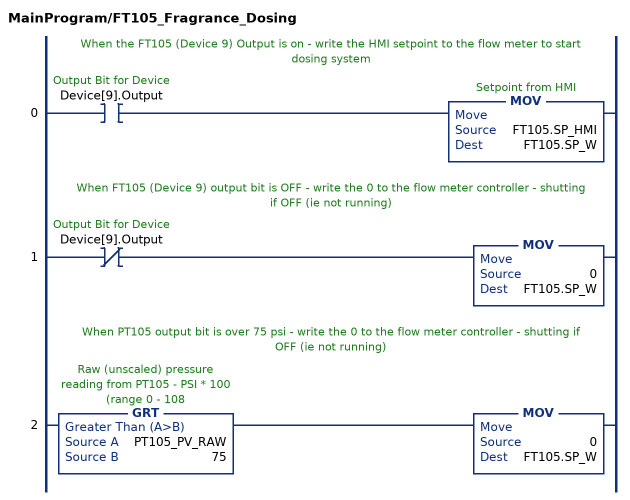
   // When the FT105 (Device 9) Output is on - write the HMI setpoint to the flow meter to start dosing system
   0: XIC(Device[9].Output)MOV(FT105.SP_HMI,FT105.SP_W);
   // When FT105 (Device 9) output bit is OFF - write the 0 to the flow meter controller - shutting if OFF (ie not running)
   1: XIO(Device[9].Output)MOV(0,FT105.SP_W);
   // When PT105 output bit is over 75 psi - write the 0 to the flow meter controller - shutting if OFF (ie not running)
   2: GRT(PT105_PV_RAW,75)MOV(0,FT105.SP_W);
END_ROUTINE

ROUTINE GF101_Thayer1_WB_Feeder   (* ladder *)
// Thayer1 WB Feeder Control Logic (Old Limestone Feeder) - not associated with Device Iteration Logic
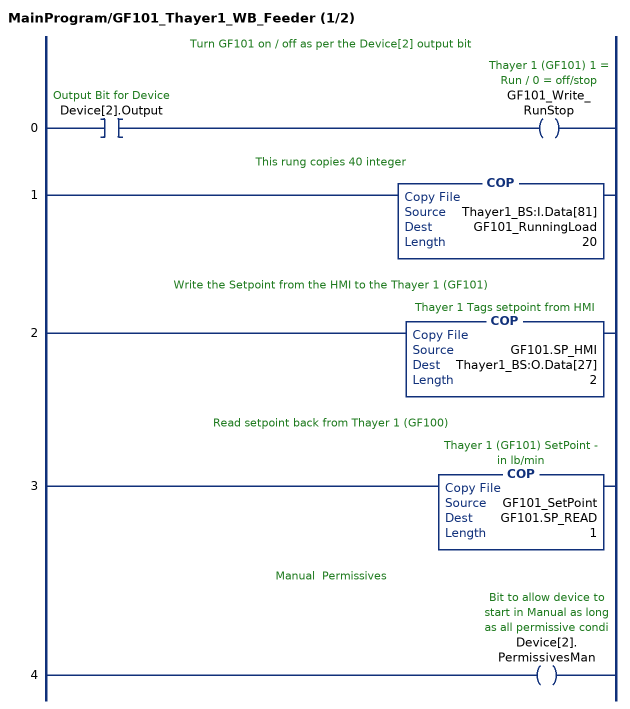
   // Turn GF101 on / off as per the Device[2] output bit
   0: XIC(Device[2].Output)OTE(GF101_Write_RunStop);
   // This rung copies 40 integer
   1: COP(Thayer1_BS:I.Data[81],GF101_RunningLoad,20);
   // Write the Setpoint from the HMI to the Thayer 1 (GF101)
   2: COP(GF101.SP_HMI,Thayer1_BS:O.Data[27],2);
   // Read setpoint back from Thayer 1 (GF100)
   3: COP(GF101_SetPoint,GF101.SP_READ,1);
   // Manual  Permissives
   4: OTE(Device[2].PermissivesMan);
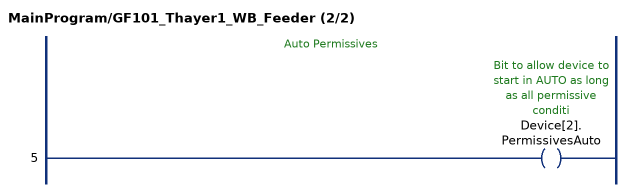
   // Auto Permissives
   5: OTE(Device[2].PermissivesAuto);
END_ROUTINE

ROUTINE GF201_Thayer2_WB_Feeder   (* ladder *)
// Thayer2 WB Feeder Control Logic (Old - Bentonite Feeder) not associated with Device Iteration Logic
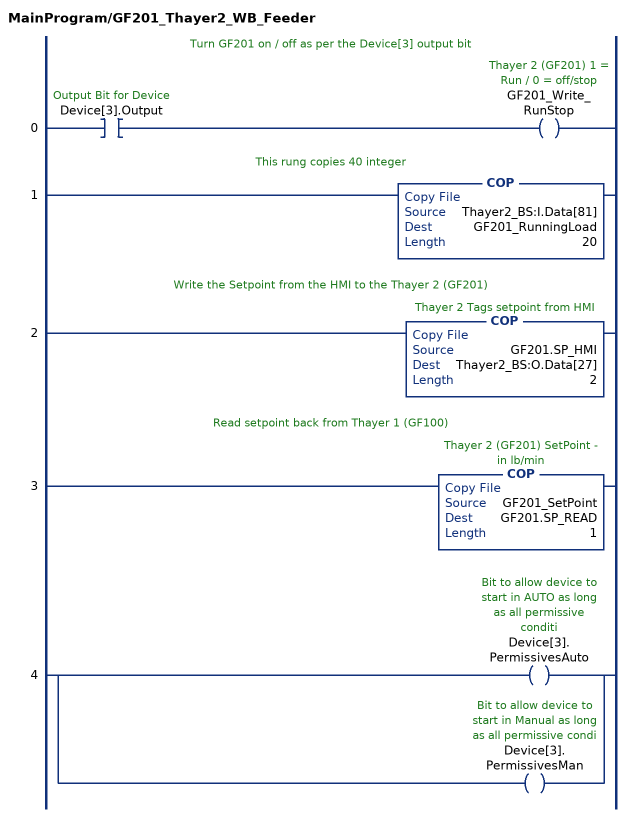
   // Turn GF201 on / off as per the Device[3] output bit
   0: XIC(Device[3].Output)OTE(GF201_Write_RunStop);
   // This rung copies 40 integer
   1: COP(Thayer2_BS:I.Data[81],GF201_RunningLoad,20);
   // Write the Setpoint from the HMI to the Thayer 2 (GF201)
   2: COP(GF201.SP_HMI,Thayer2_BS:O.Data[27],2);
   // Read setpoint back from Thayer 1 (GF100)
   3: COP(GF201_SetPoint,GF201.SP_READ,1);
   4: [OTE(Device[3].PermissivesAuto) ,OTE(Device[3].PermissivesMan) ];
END_ROUTINE

ROUTINE GF201Dose   (* ladder *)
// Logic to Dose a specific amount from GF201 - Thayer 2
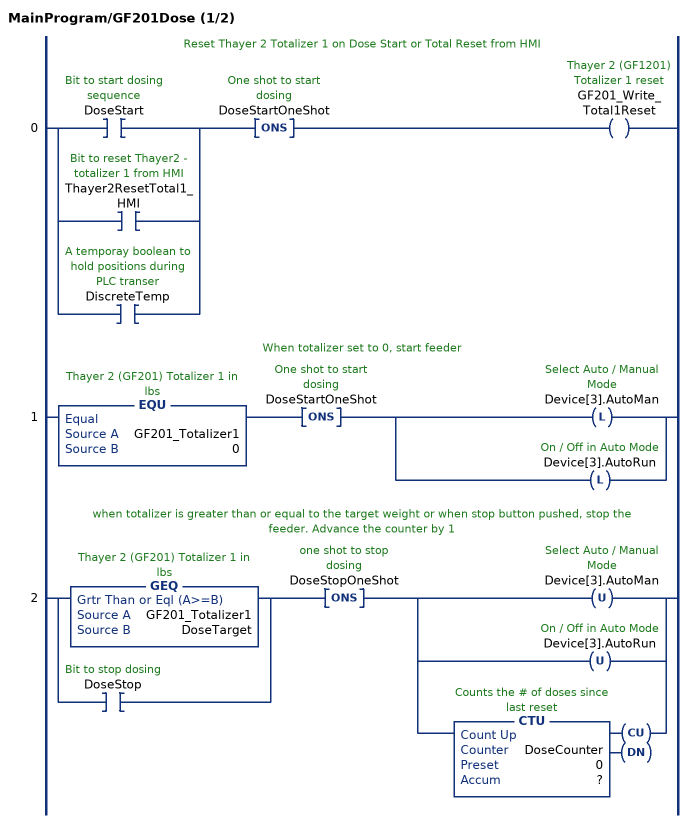
   // Reset Thayer 2 Totalizer 1 on Dose Start or Total Reset from HMI
   0: [XIC(DoseStart) ,[XIC(Thayer2ResetTotal1_HMI) ,XIC(DiscreteTemp) ] ]ONS(DoseStartOneShot)OTE(GF201_Write_Total1Reset);
   // When totalizer set to 0, start feeder
   1: EQU(GF201_Totalizer1,0)ONS(DoseStartOneShot)[OTL(Device[3].AutoMan) ,OTL(Device[3].AutoRun) ];
   // when totalizer is greater than or equal to the target weight or when stop button pushed, stop the feeder. Advance the counter by 1
   2: [GEQ(GF201_Totalizer1,DoseTarget) ,XIC(DoseStop) ]ONS(DoseStopOneShot)[OTU(Device[3].AutoMan) ,[OTU(Device[3].AutoRun) ,CTU(DoseCounter,?,?) ] ];
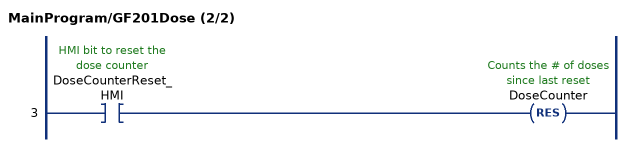
   3: XIC(DoseCounterReset_HMI)RES(DoseCounter);
END_ROUTINE

ROUTINE GF301_Small_Feeder_AcrisonLIW   (* ladder *)
// Small Feeder 1 Control via Acrison Drive SBC 2000 - not associated with Device Iteration Logic
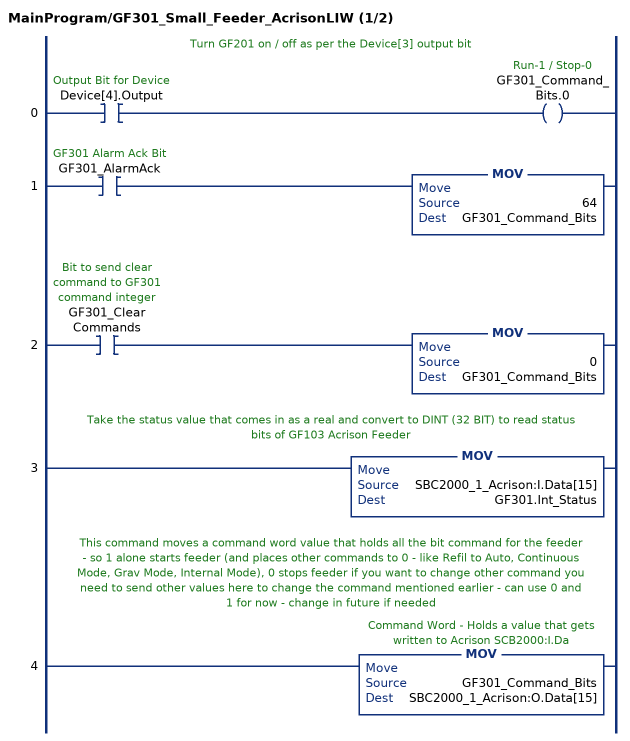
   // Turn GF201 on / off as per the Device[3] output bit
   0: XIC(Device[4].Output)OTE(GF301_Command_Bits.0);
   1: XIC(GF301_AlarmAck)MOV(64,GF301_Command_Bits);
   2: XIC(GF301_ClearCommands)MOV(0,GF301_Command_Bits);
   // Take the status value that comes in as a real and convert to DINT (32 BIT) to read status bits of GF103 Acrison Feeder
   3: MOV(SBC2000_1_Acrison:I.Data[15],GF301.Int_Status);
   // This command moves a command word value that holds all the bit command for the feeder - so 1 alone starts feeder (and places other commands to 0 - like Refil to Auto, Continuous Mode, Grav Mode, Internal Mode), 0 stops feeder if you want to change other command you need to send other values here to change the command mentioned earlier - can use 0 and 1 for now - change in future if needed
   4: MOV(GF301_Command_Bits,SBC2000_1_Acrison:O.Data[15]);
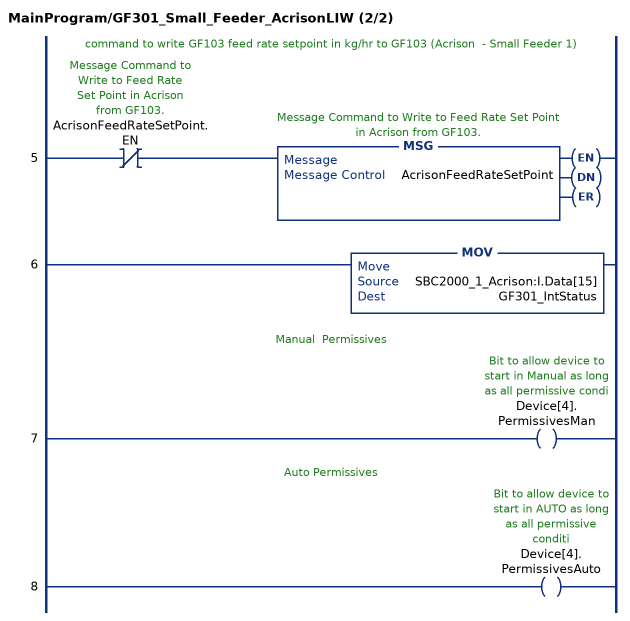
   // command to write GF103 feed rate setpoint in kg/hr to GF103 (Acrison  - Small Feeder 1)
   5: XIO(AcrisonFeedRateSetPoint.EN)MSG(AcrisonFeedRateSetPoint);
   6: MOV(SBC2000_1_Acrison:I.Data[15],GF301_IntStatus);
   // Manual  Permissives
   7: OTE(Device[4].PermissivesMan);
   // Auto Permissives
   8: OTE(Device[4].PermissivesAuto);
END_ROUTINE

ROUTINE Initialize   (* ladder *)
// Reset controls and any other initialization required
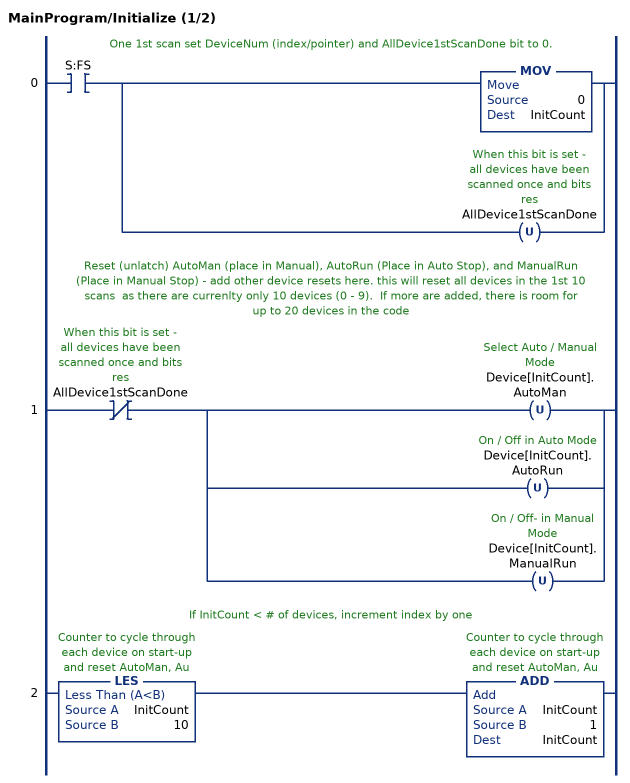
   // One 1st scan set DeviceNum (index/pointer) and AllDevice1stScanDone bit to 0.
   0: XIC(S:FS)[MOV(0,InitCount) ,OTU(AllDevice1stScanDone) ];
   // Reset (unlatch) AutoMan (place in Manual), AutoRun (Place in Auto Stop), and ManualRun (Place in Manual Stop) - add other device resets here. this will reset all devices in the 1st 10 scans  as there are currenlty only 10 devices (0 - 9).  If more are added, there is room for up to 20 devices in the code
   1: XIO(AllDevice1stScanDone)[OTU(Device[InitCount].AutoMan) ,[OTU(Device[InitCount].AutoRun) ,OTU(Device[InitCount].ManualRun) ] ];
   // If InitCount < # of devices, increment index by one
   2: LES(InitCount,10)ADD(InitCount,1,InitCount);
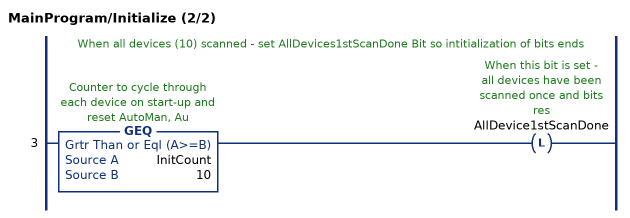
   // When all devices (10) scanned - set AllDevices1stScanDone Bit so intitialization of bits ends
   3: GEQ(InitCount,10)OTL(AllDevice1stScanDone);
END_ROUTINE
